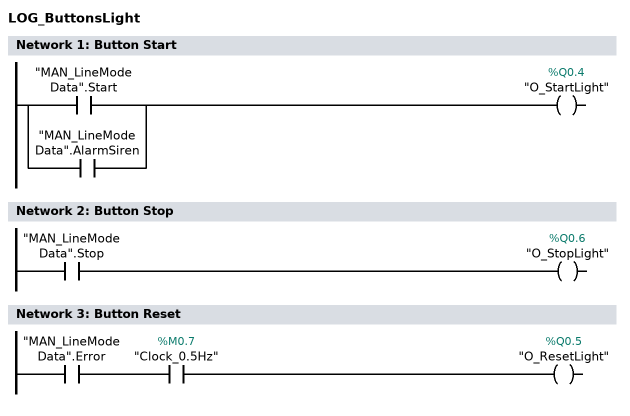
   RUNG wire#powerrail
      Contact( "MAN_LineModeData".Start )
      wire#w1
      Coil( "O_StartLight" )
   END_RUNG
   RUNG wire#powerrail
      Contact( "MAN_LineModeData".AlarmSiren )
   END_RUNG wire#w1
   // the same network as SCL:
   "O_StartLight" := "MAN_LineModeData".Start OR "MAN_LineModeData".AlarmSiren;
END_REGION

REGION Network 2: Button Stop
   RUNG wire#powerrail
      Contact( "MAN_LineModeData".Stop )
      Coil( "O_StopLight" )
   END_RUNG
   // the same network as SCL:
   "O_StopLight" := "MAN_LineModeData".Stop;
END_REGION

REGION Network 3: Button Reset
   RUNG wire#powerrail
      Contact( "MAN_LineModeData".Error )
      Contact( "Clock_0.5Hz" )
      Coil( "O_ResetLight" )
   END_RUNG
   // the same network as SCL:
   "O_ResetLight" := "MAN_LineModeData".Error AND "Clock_0.5Hz";
END_REGION
END_FUNCTION

FUNCTION "LOG_ButtonsManualLight" : Void   // FC15, LAD
{ S7_Optimized_Access := 'TRUE' }
VERSION : 0.1
// stored: AutoNumber true, IsIECCheckEnabled false, SetENOAutomatically false, UDAEnableTagReadback false
BEGIN

REGION Network 1: Button C1 light
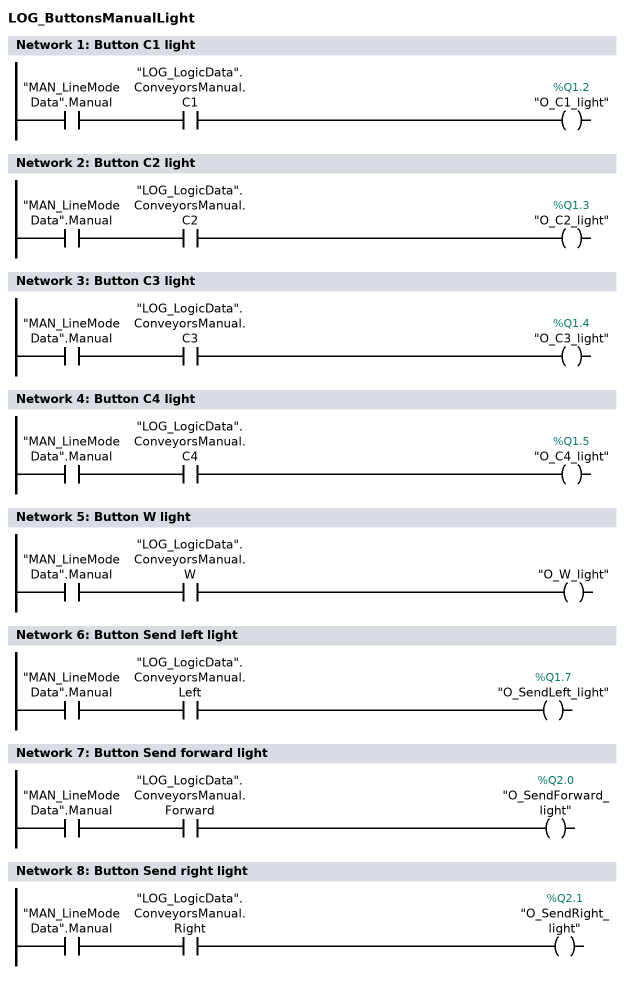
   RUNG wire#powerrail
      Contact( "MAN_LineModeData".Manual )
      Contact( "LOG_LogicData".ConveyorsManual.C1 )
      Coil( "O_C1_light" )
   END_RUNG
   // the same network as SCL:
   "O_C1_light" := "MAN_LineModeData".Manual AND "LOG_LogicData".ConveyorsManual.C1;
END_REGION

REGION Network 2: Button C2 light
   RUNG wire#powerrail
      Contact( "MAN_LineModeData".Manual )
      Contact( "LOG_LogicData".ConveyorsManual.C2 )
      Coil( "O_C2_light" )
   END_RUNG
   // the same network as SCL:
   "O_C2_light" := "MAN_LineModeData".Manual AND "LOG_LogicData".ConveyorsManual.C2;
END_REGION

REGION Network 3: Button C3 light
   RUNG wire#powerrail
      Contact( "MAN_LineModeData".Manual )
      Contact( "LOG_LogicData".ConveyorsManual.C3 )
      Coil( "O_C3_light" )
   END_RUNG
   // the same network as SCL:
   "O_C3_light" := "MAN_LineModeData".Manual AND "LOG_LogicData".ConveyorsManual.C3;
END_REGION

REGION Network 4: Button C4 light
   RUNG wire#powerrail
      Contact( "MAN_LineModeData".Manual )
      Contact( "LOG_LogicData".ConveyorsManual.C4 )
      Coil( "O_C4_light" )
   END_RUNG
   // the same network as SCL:
   "O_C4_light" := "MAN_LineModeData".Manual AND "LOG_LogicData".ConveyorsManual.C4;
END_REGION

REGION Network 5: Button W light
   RUNG wire#powerrail
      Contact( "MAN_LineModeData".Manual )
      Contact( "LOG_LogicData".ConveyorsManual.W )
      Coil( "O_W_light" )
   END_RUNG
   // the same network as SCL:
   "O_W_light" := "MAN_LineModeData".Manual AND "LOG_LogicData".ConveyorsManual.W;
END_REGION

REGION Network 6: Button Send left light
   RUNG wire#powerrail
      Contact( "MAN_LineModeData".Manual )
      Contact( "LOG_LogicData".ConveyorsManual.Left )
      Coil( "O_SendLeft_light" )
   END_RUNG
   // the same network as SCL:
   "O_SendLeft_light" := "MAN_LineModeData".Manual AND "LOG_LogicData".ConveyorsManual.Left;
END_REGION

REGION Network 7: Button Send forward light
   RUNG wire#powerrail
      Contact( "MAN_LineModeData".Manual )
      Contact( "LOG_LogicData".ConveyorsManual.Forward )
      Coil( "O_SendForward_light" )
   END_RUNG
   // the same network as SCL:
   "O_SendForward_light" := "MAN_LineModeData".Manual AND "LOG_LogicData".ConveyorsManual.Forward;
END_REGION

REGION Network 8: Button Send right light
   RUNG wire#powerrail
      Contact( "MAN_LineModeData".Manual )
      Contact( "LOG_LogicData".ConveyorsManual.Right )
      Coil( "O_SendRight_light" )
   END_RUNG
   // the same network as SCL:
   "O_SendRight_light" := "MAN_LineModeData".Manual AND "LOG_LogicData".ConveyorsManual.Right;
END_REGION
END_FUNCTION

FUNCTION "LOG_ColumnLight" : Void   // FC16, LAD
{ S7_Optimized_Access := 'TRUE' }
VERSION : 0.1
// stored: AutoNumber true, IsIECCheckEnabled false, SetENOAutomatically false, UDAEnableTagReadback false
   VAR_TEMP
      Green_1 : Bool;
      Green_2 : Bool;
      Yellow_1 : Bool;
      Yellow_2 : Bool;
   END_VAR
BEGIN

REGION Network 1: Start line manual mode signaling
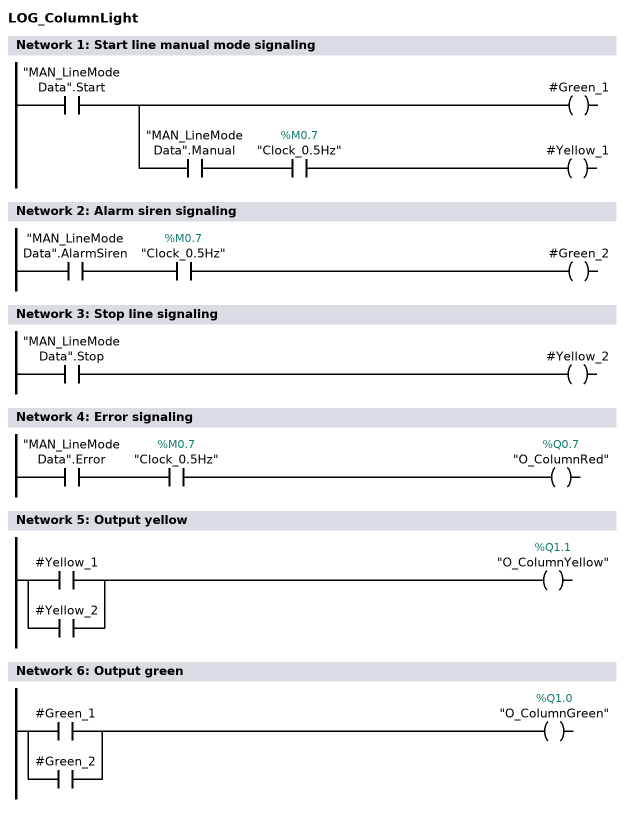
   RUNG wire#powerrail
      Contact( "MAN_LineModeData".Start )
      wire#w1
      Coil( #Green_1 )
   END_RUNG
   RUNG wire#w1
      Contact( "MAN_LineModeData".Manual )
      Contact( "Clock_0.5Hz" )
      Coil( #Yellow_1 )
   END_RUNG
   // the same network as SCL:
   #Green_1 := "MAN_LineModeData".Start;
   #Yellow_1 := "MAN_LineModeData".Start AND "MAN_LineModeData".Manual AND "Clock_0.5Hz";
END_REGION

REGION Network 2: Alarm siren signaling
   RUNG wire#powerrail
      Contact( "MAN_LineModeData".AlarmSiren )
      Contact( "Clock_0.5Hz" )
      Coil( #Green_2 )
   END_RUNG
   // the same network as SCL:
   #Green_2 := "MAN_LineModeData".AlarmSiren AND "Clock_0.5Hz";
END_REGION

REGION Network 3: Stop line signaling
   RUNG wire#powerrail
      Contact( "MAN_LineModeData".Stop )
      Coil( #Yellow_2 )
   END_RUNG
   // the same network as SCL:
   #Yellow_2 := "MAN_LineModeData".Stop;
END_REGION

REGION Network 4: Error signaling
   RUNG wire#powerrail
      Contact( "MAN_LineModeData".Error )
      Contact( "Clock_0.5Hz" )
      Coil( "O_ColumnRed" )
   END_RUNG
   // the same network as SCL:
   "O_ColumnRed" := "MAN_LineModeData".Error AND "Clock_0.5Hz";
END_REGION

REGION Network 5: Output yellow
   RUNG wire#powerrail
      Contact( #Yellow_1 )
      wire#w1
      Coil( "O_ColumnYellow" )
   END_RUNG
   RUNG wire#powerrail
      Contact( #Yellow_2 )
   END_RUNG wire#w1
   // the same network as SCL:
   "O_ColumnYellow" := #Yellow_1 OR #Yellow_2;
END_REGION

REGION Network 6: Output green
   RUNG wire#powerrail
      Contact( #Green_1 )
      wire#w1
      Coil( "O_ColumnGreen" )
   END_RUNG
   RUNG wire#powerrail
      Contact( #Green_2 )
   END_RUNG wire#w1
   // the same network as SCL:
   "O_ColumnGreen" := #Green_1 OR #Green_2;
END_REGION
END_FUNCTION

FUNCTION "LOG_Light" : Void   // FC11, LAD
{ S7_Optimized_Access := 'TRUE' }
VERSION : 0.1
// stored: AutoNumber true, IsIECCheckEnabled false, SetENOAutomatically false, UDAEnableTagReadback false
BEGIN

REGION Network 1: Call: ButtonsLight
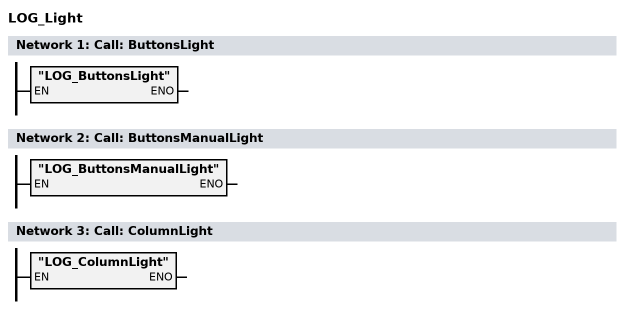
   RUNG wire#powerrail
      "LOG_ButtonsLight"()
   END_RUNG
   // the same network as SCL:
   "LOG_ButtonsLight"();
END_REGION

REGION Network 2: Call: ButtonsManualLight
   RUNG wire#powerrail
      "LOG_ButtonsManualLight"()
   END_RUNG
   // the same network as SCL:
   "LOG_ButtonsManualLight"();
END_REGION

REGION Network 3: Call: ColumnLight
   RUNG wire#powerrail
      "LOG_ColumnLight"()
   END_RUNG
   // the same network as SCL:
   "LOG_ColumnLight"();
END_REGION
END_FUNCTION

FUNCTION "LOG_Statistic" : Void   // FC8, LAD
{ S7_Optimized_Access := 'TRUE' }
VERSION : 0.1
// stored: AutoNumber false, IsIECCheckEnabled false, SetENOAutomatically false, UDAEnableTagReadback false
   VAR_TEMP
      t_RisingEdge : Bool;
   END_VAR
BEGIN

REGION Network 1: Call: CountPackages
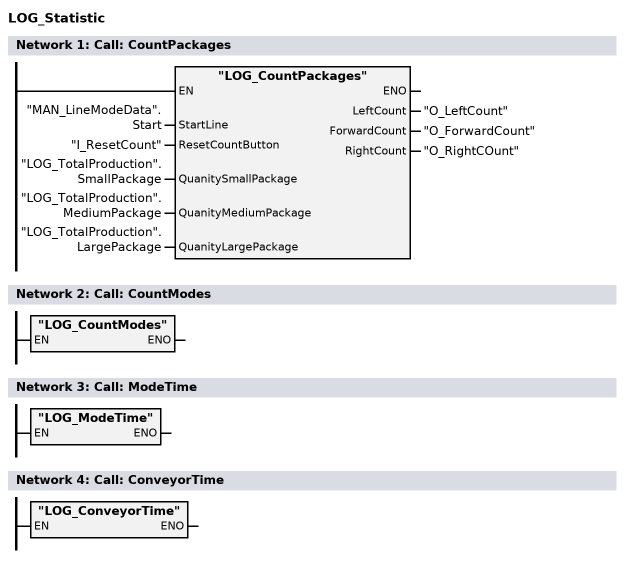
   RUNG wire#powerrail
      "LOG_CountPackages"(StartLine := "MAN_LineModeData".Start, ResetCountButton := "I_ResetCount", QuanitySmallPackage := "LOG_TotalProduction".SmallPackage, QuanityMediumPackage := "LOG_TotalProduction".MediumPackage, QuanityLargePackage := "LOG_TotalProduction".LargePackage, LeftCount => "O_LeftCount", ForwardCount => "O_ForwardCount", RightCount => "O_RightCOunt")
   END_RUNG
   // the same network as SCL:
   "LOG_CountPackages"(StartLine := "MAN_LineModeData".Start,
                       ResetCountButton := "I_ResetCount",
                       QuanitySmallPackage := "LOG_TotalProduction".SmallPackage,
                       QuanityMediumPackage := "LOG_TotalProduction".MediumPackage,
                       QuanityLargePackage := "LOG_TotalProduction".LargePackage,
                       LeftCount => "O_LeftCount",
                       ForwardCount => "O_ForwardCount",
                       RightCount => "O_RightCOunt");
END_REGION

REGION Network 2: Call: CountModes
   RUNG wire#powerrail
      "LOG_CountModes"()
   END_RUNG
   // the same network as SCL:
   "LOG_CountModes"();
END_REGION

REGION Network 3: Call: ModeTime
   RUNG wire#powerrail
      "LOG_ModeTime"()
   END_RUNG
   // the same network as SCL:
   "LOG_ModeTime"();
END_REGION

REGION Network 4: Call: ConveyorTime
   RUNG wire#powerrail
      "LOG_ConveyorTime"()
   END_RUNG
   // the same network as SCL:
   "LOG_ConveyorTime"();
END_REGION
END_FUNCTION

FUNCTION "LOG_CountPackages" : Void   // FC9, LAD
{ S7_Optimized_Access := 'TRUE' }
VERSION : 0.1
// stored: AutoNumber false, IsIECCheckEnabled false, SetENOAutomatically false, UDAEnableTagReadback false
   VAR_INPUT
      StartLine : Bool;
      ResetCountButton : Bool;
   END_VAR
   VAR_OUTPUT
      LeftCount : Int;
      ForwardCount : Int;
      RightCount : Int;
   END_VAR
   VAR_IN_OUT
      QuanitySmallPackage : Int;
      QuanityMediumPackage : Int;
      QuanityLargePackage : Int;
   END_VAR
BEGIN

REGION Network 1
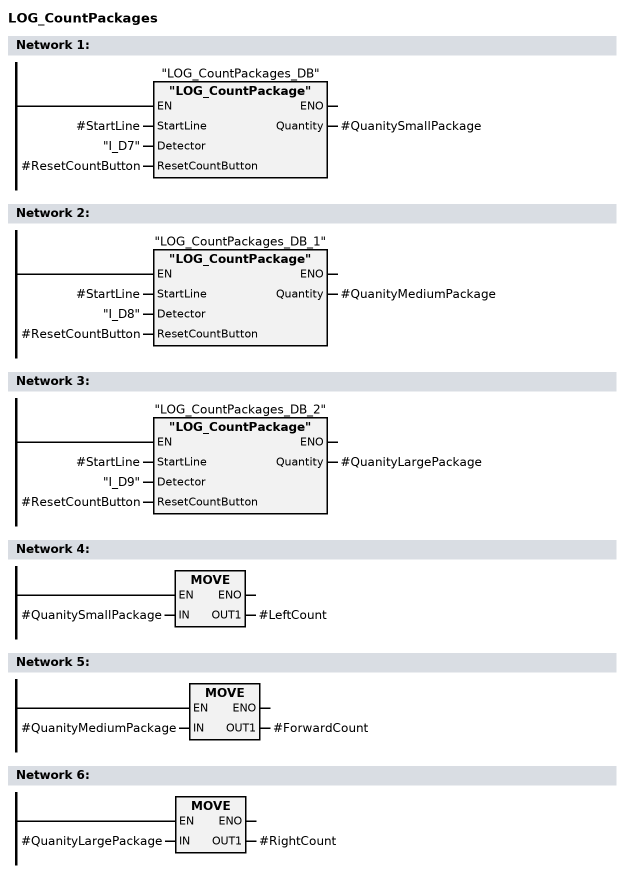
   RUNG wire#powerrail
      "LOG_CountPackages_DB"(StartLine := #StartLine, Detector := "I_D7", ResetCountButton := #ResetCountButton, Quantity => #QuanitySmallPackage)
   END_RUNG
   // the same network as SCL:
   "LOG_CountPackages_DB"(StartLine := #StartLine,   // "LOG_CountPackage"
                          Detector := "I_D7",
                          ResetCountButton := #ResetCountButton,
                          Quantity => #QuanitySmallPackage);
END_REGION

REGION Network 2
   RUNG wire#powerrail
      "LOG_CountPackages_DB_1"(StartLine := #StartLine, Detector := "I_D8", ResetCountButton := #ResetCountButton, Quantity => #QuanityMediumPackage)
   END_RUNG
   // the same network as SCL:
   "LOG_CountPackages_DB_1"(StartLine := #StartLine,   // "LOG_CountPackage"
                           Detector := "I_D8",
                           ResetCountButton := #ResetCountButton,
                           Quantity => #QuanityMediumPackage);
END_REGION

REGION Network 3
   RUNG wire#powerrail
      "LOG_CountPackages_DB_2"(StartLine := #StartLine, Detector := "I_D9", ResetCountButton := #ResetCountButton, Quantity => #QuanityLargePackage)
   END_RUNG
   // the same network as SCL:
   "LOG_CountPackages_DB_2"(StartLine := #StartLine,   // "LOG_CountPackage"
                           Detector := "I_D9",
                           ResetCountButton := #ResetCountButton,
                           Quantity => #QuanityLargePackage);
END_REGION

REGION Network 4
   RUNG wire#powerrail
      Move(in := #QuanitySmallPackage, out1 => #LeftCount)
   END_RUNG
   // the same network as SCL:
   #LeftCount := #QuanitySmallPackage;
END_REGION

REGION Network 5
   RUNG wire#powerrail
      Move(in := #QuanityMediumPackage, out1 => #ForwardCount)
   END_RUNG
   // the same network as SCL:
   #ForwardCount := #QuanityMediumPackage;
END_REGION

REGION Network 6
   RUNG wire#powerrail
      Move(in := #QuanityLargePackage, out1 => #RightCount)
   END_RUNG
   // the same network as SCL:
   #RightCount := #QuanityLargePackage;
END_REGION
END_FUNCTION

FUNCTION_BLOCK "LOG_CountPackage"   // FB4, LAD
{ S7_Optimized_Access := 'TRUE' }
VERSION : 0.1
// stored: AutoNumber true, IsIECCheckEnabled false, IsRetainMemResEnabled false, MemoryReserve 100, SetENOAutomatically false, UDAEnableTagReadback false
   VAR_INPUT
      StartLine : Bool;
      Detector : Bool;
      ResetCountButton : Bool;
   END_VAR
   VAR_OUTPUT
      Quantity : Int;
   END_VAR
   VAR RETAIN
      IEC_Counter_0_Instance { ExternalAccessible := 'False'; ExternalVisible := 'False'; ExternalWritable := 'False'} : CTU_INT;
      N_Detector { S7_SetPoint := 'True'} : Bool;
   END_VAR
   VAR_TEMP   // added for the SCL form of the ladder/FBD networks
      _w1 : Bool;
   END_VAR
BEGIN

REGION Network 1
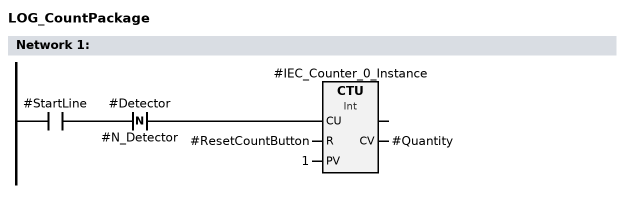
   RUNG wire#powerrail
      Contact( #StartLine )
      N_Contact(operand := #Detector, bit := #N_Detector)
      { S7_Templates := "value_type := Int" } #IEC_Counter_0_Instance.CTU(r := #ResetCountButton, pv := 1, cv => #Quantity)
   END_RUNG
   // the same network as SCL:
   #_w1 := #StartLine AND NOT #Detector AND #N_Detector;   // falling edge of #Detector
   #N_Detector := #Detector;
   #IEC_Counter_0_Instance(CU := #_w1, R := #ResetCountButton, PV := 1, CV => #Quantity);   // CTU
END_REGION
END_FUNCTION_BLOCK

FUNCTION "LOG_CountModes" : Void   // FC19, LAD
{ S7_Optimized_Access := 'TRUE' }
VERSION : 0.1
// stored: AutoNumber true, IsIECCheckEnabled false, SetENOAutomatically false, UDAEnableTagReadback false
BEGIN

REGION Network 1: Call: CountMode - Auto
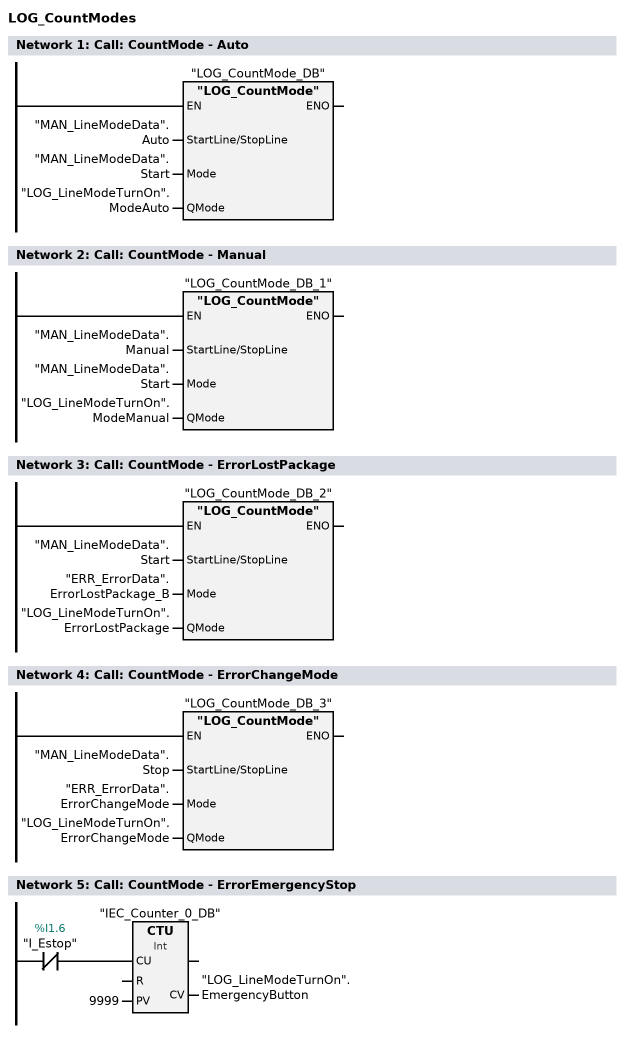
   RUNG wire#powerrail
      "LOG_CountMode_DB"("StartLine/StopLine" := "MAN_LineModeData".Auto, Mode := "MAN_LineModeData".Start, QMode := "LOG_LineModeTurnOn".ModeAuto)
   END_RUNG
   // the same network as SCL:
   "LOG_CountMode_DB"("StartLine/StopLine" := "MAN_LineModeData".Auto,   // "LOG_CountMode"
                      Mode := "MAN_LineModeData".Start,
                      QMode := "LOG_LineModeTurnOn".ModeAuto);
END_REGION

REGION Network 2: Call: CountMode - Manual
   RUNG wire#powerrail
      "LOG_CountMode_DB_1"("StartLine/StopLine" := "MAN_LineModeData".Manual, Mode := "MAN_LineModeData".Start, QMode := "LOG_LineModeTurnOn".ModeManual)
   END_RUNG
   // the same network as SCL:
   "LOG_CountMode_DB_1"("StartLine/StopLine" := "MAN_LineModeData".Manual,   // "LOG_CountMode"
                        Mode := "MAN_LineModeData".Start,
                        QMode := "LOG_LineModeTurnOn".ModeManual);
END_REGION

REGION Network 3: Call: CountMode - ErrorLostPackage
   RUNG wire#powerrail
      "LOG_CountMode_DB_2"("StartLine/StopLine" := "MAN_LineModeData".Start, Mode := "ERR_ErrorData".ErrorLostPackage_B, QMode := "LOG_LineModeTurnOn".ErrorLostPackage)
   END_RUNG
   // the same network as SCL:
   "LOG_CountMode_DB_2"("StartLine/StopLine" := "MAN_LineModeData".Start,   // "LOG_CountMode"
                        Mode := "ERR_ErrorData".ErrorLostPackage_B,
                        QMode := "LOG_LineModeTurnOn".ErrorLostPackage);
END_REGION

REGION Network 4: Call: CountMode - ErrorChangeMode
   RUNG wire#powerrail
      "LOG_CountMode_DB_3"("StartLine/StopLine" := "MAN_LineModeData".Stop, Mode := "ERR_ErrorData".ErrorChangeMode, QMode := "LOG_LineModeTurnOn".ErrorChangeMode)
   END_RUNG
   // the same network as SCL:
   "LOG_CountMode_DB_3"("StartLine/StopLine" := "MAN_LineModeData".Stop,   // "LOG_CountMode"
                        Mode := "ERR_ErrorData".ErrorChangeMode,
                        QMode := "LOG_LineModeTurnOn".ErrorChangeMode);
END_REGION

REGION Network 5: Call: CountMode - ErrorEmergencyStop
   RUNG wire#powerrail
      I_Contact( "I_Estop" )
      { S7_Templates := "value_type := Int" } "IEC_Counter_0_DB".CTU(r :=, pv := 9999, cv => "LOG_LineModeTurnOn".EmergencyButton)
   END_RUNG
   // the same network as SCL:
   "IEC_Counter_0_DB".CTU(CU := NOT "I_Estop", PV := 9999, CV => "LOG_LineModeTurnOn".EmergencyButton);
END_REGION
END_FUNCTION

FUNCTION_BLOCK "LOG_CountMode"   // FB3, LAD
{ S7_Optimized_Access := 'TRUE' }
VERSION : 0.1
// stored: AutoNumber true, IsIECCheckEnabled false, IsRetainMemResEnabled false, MemoryReserve 100, SetENOAutomatically false, UDAEnableTagReadback false
   VAR_INPUT
      "StartLine/StopLine" : Bool;
      Mode : Bool;
   END_VAR
   VAR_IN_OUT
      QMode : UDInt;
   END_VAR
   VAR
      P_Mode : Bool;
   END_VAR
   VAR_TEMP   // added for the SCL form of the ladder/FBD networks
      _w1 : Bool;
   END_VAR
BEGIN

REGION Network 1
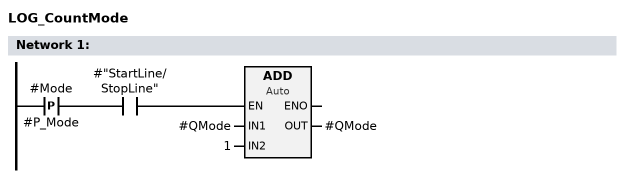
   RUNG wire#powerrail
      P_Contact(operand := #Mode, bit := #P_Mode)
      Contact( #"StartLine/StopLine" )
      { S7_GenerateENO := "TRUE" } Add(in1 := #QMode, in2 := 1, out => #QMode)
   END_RUNG
   // the same network as SCL:
   #_w1 := #Mode AND NOT #P_Mode;   // rising edge of #Mode
   #P_Mode := #Mode;
   IF #_w1 AND #"StartLine/StopLine" THEN #QMode := #QMode + 1; END_IF;
END_REGION
END_FUNCTION_BLOCK

FUNCTION "LOG_ModeTime" : Void   // FC18, LAD
{ S7_Optimized_Access := 'TRUE' }
VERSION : 0.1
// stored: AutoNumber true, IsIECCheckEnabled false, SetENOAutomatically false, UDAEnableTagReadback false
   VAR_TEMP
      t_RisingEdge : Bool;
   END_VAR
BEGIN

REGION Network 1: Trigger
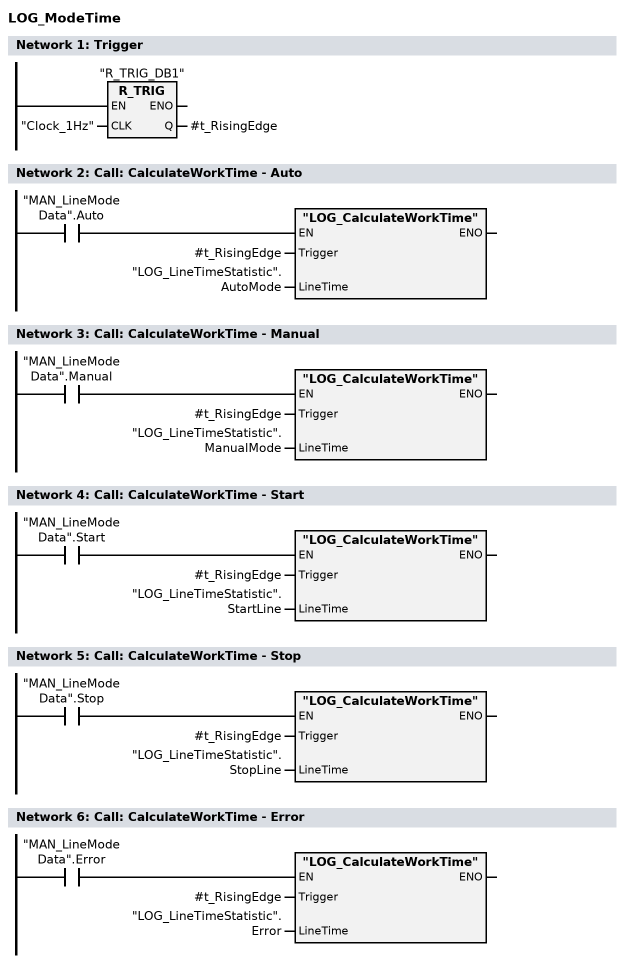
   RUNG wire#powerrail
      "R_TRIG_DB1".R_TRIG(CLK := "Clock_1Hz", Q => #t_RisingEdge)
   END_RUNG
   // the same network as SCL:
   "R_TRIG_DB1"(CLK := "Clock_1Hz", Q => #t_RisingEdge);   // R_TRIG
END_REGION

REGION Network 2: Call: CalculateWorkTime - Auto
   RUNG wire#powerrail
      Contact( "MAN_LineModeData".Auto )
      "LOG_CalculateWorkTime"(Trigger := #t_RisingEdge, LineTime := "LOG_LineTimeStatistic".AutoMode)
   END_RUNG
   // the same network as SCL:
   IF "MAN_LineModeData".Auto THEN
       "LOG_CalculateWorkTime"(Trigger := #t_RisingEdge, LineTime := "LOG_LineTimeStatistic".AutoMode);
   END_IF;
END_REGION

REGION Network 3: Call: CalculateWorkTime - Manual
   RUNG wire#powerrail
      Contact( "MAN_LineModeData".Manual )
      "LOG_CalculateWorkTime"(Trigger := #t_RisingEdge, LineTime := "LOG_LineTimeStatistic".ManualMode)
   END_RUNG
   // the same network as SCL:
   IF "MAN_LineModeData".Manual THEN
       "LOG_CalculateWorkTime"(Trigger := #t_RisingEdge, LineTime := "LOG_LineTimeStatistic".ManualMode);
   END_IF;
END_REGION

REGION Network 4: Call: CalculateWorkTime - Start
   RUNG wire#powerrail
      Contact( "MAN_LineModeData".Start )
      "LOG_CalculateWorkTime"(Trigger := #t_RisingEdge, LineTime := "LOG_LineTimeStatistic".StartLine)
   END_RUNG
   // the same network as SCL:
   IF "MAN_LineModeData".Start THEN
       "LOG_CalculateWorkTime"(Trigger := #t_RisingEdge, LineTime := "LOG_LineTimeStatistic".StartLine);
   END_IF;
END_REGION

REGION Network 5: Call: CalculateWorkTime - Stop
   RUNG wire#powerrail
      Contact( "MAN_LineModeData".Stop )
      "LOG_CalculateWorkTime"(Trigger := #t_RisingEdge, LineTime := "LOG_LineTimeStatistic".StopLine)
   END_RUNG
   // the same network as SCL:
   IF "MAN_LineModeData".Stop THEN
       "LOG_CalculateWorkTime"(Trigger := #t_RisingEdge, LineTime := "LOG_LineTimeStatistic".StopLine);
   END_IF;
END_REGION

REGION Network 6: Call: CalculateWorkTime - Error
   RUNG wire#powerrail
      Contact( "MAN_LineModeData".Error )
      "LOG_CalculateWorkTime"(Trigger := #t_RisingEdge, LineTime := "LOG_LineTimeStatistic".Error)
   END_RUNG
   // the same network as SCL:
   IF "MAN_LineModeData".Error THEN
       "LOG_CalculateWorkTime"(Trigger := #t_RisingEdge, LineTime := "LOG_LineTimeStatistic".Error);
   END_IF;
END_REGION
END_FUNCTION

FUNCTION "LOG_CalculateWorkTime" : Void   // FC1300, LAD
{ S7_Optimized_Access := 'TRUE' }
VERSION : 0.1
// stored: AutoNumber false, IsIECCheckEnabled false, SetENOAutomatically false, UDAEnableTagReadback false
   VAR_INPUT
      Trigger : Bool;
   END_VAR
   VAR_IN_OUT
      LineTime : "stt_TimeWork";
   END_VAR
   VAR_TEMP   // added for the SCL form of the ladder/FBD networks
      _w1 : Bool;
   END_VAR
BEGIN

REGION Network 1: Seconds
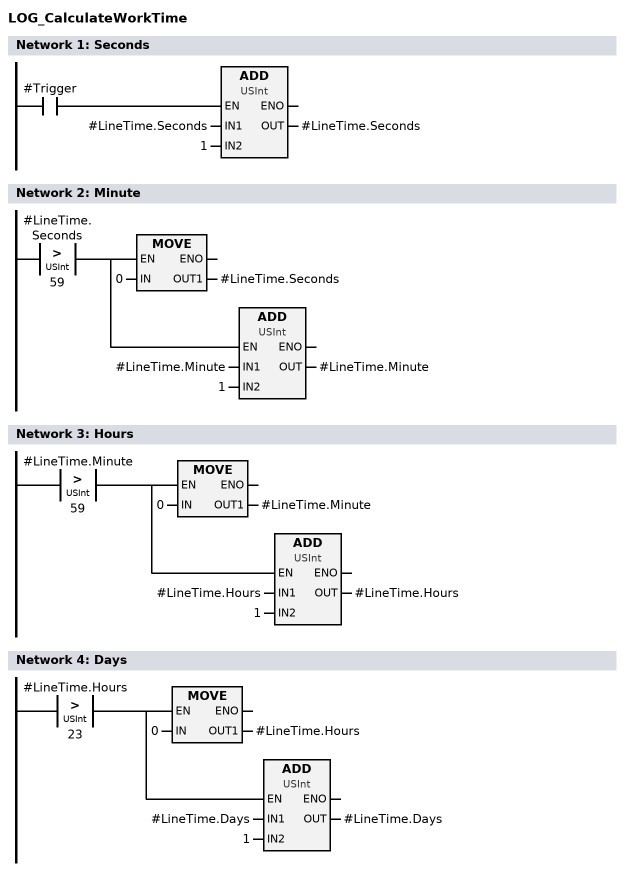
   RUNG wire#powerrail
      Contact( #Trigger )
      { S7_Templates := "SrcType := USInt"; S7_GenerateENO := "TRUE" } Add(in1 := #LineTime.Seconds, in2 := 1, out => #LineTime.Seconds)
   END_RUNG
   // the same network as SCL:
   IF #Trigger THEN #LineTime.Seconds := #LineTime.Seconds + 1; END_IF;
END_REGION

REGION Network 2: Minute
   RUNG wire#powerrail
      { S7_Templates := "SrcType := USInt" } GT_Contact(in1 := #LineTime.Seconds, in2 := 59)
      wire#w1
      { S7_GenerateENO := "TRUE" } Move(in := 0, out1 => #LineTime.Seconds)
   END_RUNG
   RUNG wire#w1
      { S7_Templates := "SrcType := USInt"; S7_GenerateENO := "TRUE" } Add(in1 := #LineTime.Minute, in2 := 1, out => #LineTime.Minute)
   END_RUNG
   // the same network as SCL:
   #_w1 := #LineTime.Seconds > 59;
   IF #_w1 THEN
       #LineTime.Seconds := 0;
       #LineTime.Minute := #LineTime.Minute + 1;
   END_IF;
END_REGION

REGION Network 3: Hours
   RUNG wire#powerrail
      { S7_Templates := "SrcType := USInt" } GT_Contact(in1 := #LineTime.Minute, in2 := 59)
      wire#w1
      { S7_GenerateENO := "TRUE" } Move(in := 0, out1 => #LineTime.Minute)
   END_RUNG
   RUNG wire#w1
      { S7_Templates := "SrcType := USInt"; S7_GenerateENO := "TRUE" } Add(in1 := #LineTime.Hours, in2 := 1, out => #LineTime.Hours)
   END_RUNG
   // the same network as SCL:
   #_w1 := #LineTime.Minute > 59;
   IF #_w1 THEN
       #LineTime.Minute := 0;
       #LineTime.Hours := #LineTime.Hours + 1;
   END_IF;
END_REGION

REGION Network 4: Days
   RUNG wire#powerrail
      { S7_Templates := "SrcType := USInt" } GT_Contact(in1 := #LineTime.Hours, in2 := 23)
      wire#w1
      { S7_GenerateENO := "TRUE" } Move(in := 0, out1 => #LineTime.Hours)
   END_RUNG
   RUNG wire#w1
      { S7_Templates := "SrcType := USInt"; S7_GenerateENO := "TRUE" } Add(in1 := #LineTime.Days, in2 := 1, out => #LineTime.Days)
   END_RUNG
   // the same network as SCL:
   #_w1 := #LineTime.Hours > 23;
   IF #_w1 THEN
       #LineTime.Hours := 0;
       #LineTime.Days := #LineTime.Days + 1;
   END_IF;
END_REGION
END_FUNCTION

FUNCTION "LOG_ConveyorTime" : Void   // FC20, LAD
{ S7_Optimized_Access := 'TRUE' }
VERSION : 0.1
// stored: AutoNumber true, IsIECCheckEnabled false, SetENOAutomatically false, UDAEnableTagReadback false
   VAR_TEMP
      t_RisingTime : Bool;
   END_VAR
BEGIN

REGION Network 1: Trigger
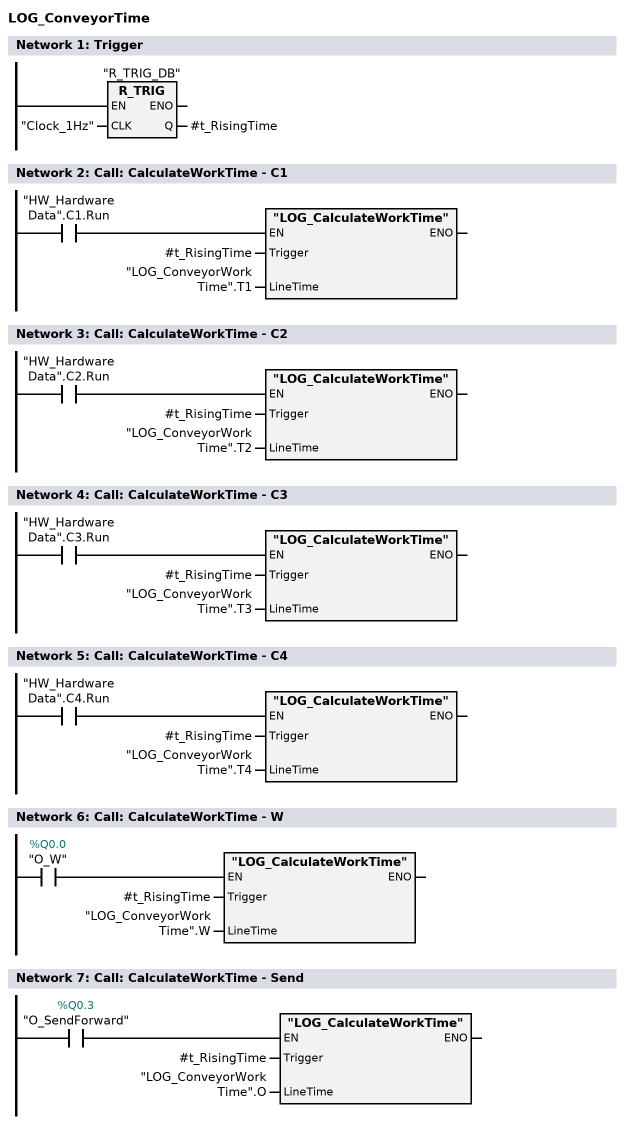
   RUNG wire#powerrail
      "R_TRIG_DB".R_TRIG(CLK := "Clock_1Hz", Q => #t_RisingTime)
   END_RUNG
   // the same network as SCL:
   "R_TRIG_DB"(CLK := "Clock_1Hz", Q => #t_RisingTime);   // R_TRIG
END_REGION

REGION Network 2: Call: CalculateWorkTime - C1
   RUNG wire#powerrail
      Contact( "HW_HardwareData".C1.Run )
      "LOG_CalculateWorkTime"(Trigger := #t_RisingTime, LineTime := "LOG_ConveyorWorkTime".T1)
   END_RUNG
   // the same network as SCL:
   IF "HW_HardwareData".C1.Run THEN
       "LOG_CalculateWorkTime"(Trigger := #t_RisingTime, LineTime := "LOG_ConveyorWorkTime".T1);
   END_IF;
END_REGION

REGION Network 3: Call: CalculateWorkTime - C2
   RUNG wire#powerrail
      Contact( "HW_HardwareData".C2.Run )
      "LOG_CalculateWorkTime"(Trigger := #t_RisingTime, LineTime := "LOG_ConveyorWorkTime".T2)
   END_RUNG
   // the same network as SCL:
   IF "HW_HardwareData".C2.Run THEN
       "LOG_CalculateWorkTime"(Trigger := #t_RisingTime, LineTime := "LOG_ConveyorWorkTime".T2);
   END_IF;
END_REGION

REGION Network 4: Call: CalculateWorkTime - C3
   RUNG wire#powerrail
      Contact( "HW_HardwareData".C3.Run )
      "LOG_CalculateWorkTime"(Trigger := #t_RisingTime, LineTime := "LOG_ConveyorWorkTime".T3)
   END_RUNG
   // the same network as SCL:
   IF "HW_HardwareData".C3.Run THEN
       "LOG_CalculateWorkTime"(Trigger := #t_RisingTime, LineTime := "LOG_ConveyorWorkTime".T3);
   END_IF;
END_REGION

REGION Network 5: Call: CalculateWorkTime - C4
   RUNG wire#powerrail
      Contact( "HW_HardwareData".C4.Run )
      "LOG_CalculateWorkTime"(Trigger := #t_RisingTime, LineTime := "LOG_ConveyorWorkTime".T4)
   END_RUNG
   // the same network as SCL:
   IF "HW_HardwareData".C4.Run THEN
       "LOG_CalculateWorkTime"(Trigger := #t_RisingTime, LineTime := "LOG_ConveyorWorkTime".T4);
   END_IF;
END_REGION

REGION Network 6: Call: CalculateWorkTime - W
   RUNG wire#powerrail
      Contact( "O_W" )
      "LOG_CalculateWorkTime"(Trigger := #t_RisingTime, LineTime := "LOG_ConveyorWorkTime".W)
   END_RUNG
   // the same network as SCL:
   IF "O_W" THEN
       "LOG_CalculateWorkTime"(Trigger := #t_RisingTime, LineTime := "LOG_ConveyorWorkTime".W);
   END_IF;
END_REGION

REGION Network 7: Call: CalculateWorkTime - Send
   RUNG wire#powerrail
      Contact( "O_SendForward" )
      "LOG_CalculateWorkTime"(Trigger := #t_RisingTime, LineTime := "LOG_ConveyorWorkTime".O)
   END_RUNG
   // the same network as SCL:
   IF "O_SendForward" THEN
       "LOG_CalculateWorkTime"(Trigger := #t_RisingTime, LineTime := "LOG_ConveyorWorkTime".O);
   END_IF;
END_REGION
END_FUNCTION

DATA_BLOCK "ERR_ChangeMode_DB"   // DB23
VERSION : 0.1
// stored: AutoNumber true, InstanceOfName ERR_ChangeMode, InstanceOfType FB
"ERR_ChangeMode"
BEGIN
END_DATA_BLOCK

DATA_BLOCK "ERR_EStop_DB"   // DB21
VERSION : 0.1
// stored: AutoNumber true, InstanceOfName ERR_EStop, InstanceOfType FB
"ERR_EStop"
BEGIN
END_DATA_BLOCK

DATA_BLOCK "HW_MotorControle_DB"   // DB6
VERSION : 0.1
// stored: AutoNumber true, InstanceOfName HW_MotorControle, InstanceOfType FB
"HW_MotorControle"
BEGIN
END_DATA_BLOCK

DATA_BLOCK "HW_MotorControle_DB_1"   // DB8
VERSION : 0.1
// stored: AutoNumber true, InstanceOfName HW_MotorControle, InstanceOfType FB
"HW_MotorControle"
BEGIN
END_DATA_BLOCK

DATA_BLOCK "HW_MotorControle_DB_2"   // DB9
VERSION : 0.1
// stored: AutoNumber true, InstanceOfName HW_MotorControle, InstanceOfType FB
"HW_MotorControle"
BEGIN
END_DATA_BLOCK

DATA_BLOCK "HW_MotorControle_DB_3"   // DB10
VERSION : 0.1
// stored: AutoNumber true, InstanceOfName HW_MotorControle, InstanceOfType FB
"HW_MotorControle"
BEGIN
END_DATA_BLOCK

DATA_BLOCK "HW_MovingAverageFilter_DB"   // DB3
VERSION : 0.1
// stored: AutoNumber true, InstanceOfName HW_MovingAverageFilter, InstanceOfType FB
"HW_MovingAverageFilter"
BEGIN
END_DATA_BLOCK

DATA_BLOCK "IEC_Counter_0_DB"   // DB35
{ S7_Optimized_Access := 'TRUE' }
// stored: AutoNumber true, InstanceOfName IEC_COUNTER, OfSystemLibElement IEC_COUNTER, OfSystemLibVersion 1.0
"IEC_COUNTER"
   // VAR RETAIN
   //    CU : Bool;
   //    CD : Bool;
   //    R : Bool;
   //    LD : Bool;
   //    QU : Bool;
   //    QD : Bool;
   //    PV : Int;
   //    CV : Int;
   // END_VAR
BEGIN
END_DATA_BLOCK

DATA_BLOCK "LOG_AutoControle_DB"   // DB11
VERSION : 0.1
// stored: AutoNumber true, InstanceOfName LOG_AutoControle, InstanceOfType FB
"LOG_AutoControle"
BEGIN
END_DATA_BLOCK

DATA_BLOCK "LOG_CountMode_DB"   // DB31
VERSION : 0.1
// stored: AutoNumber true, InstanceOfName LOG_CountMode, InstanceOfType FB
"LOG_CountMode"
BEGIN
END_DATA_BLOCK

DATA_BLOCK "LOG_CountMode_DB_1"   // DB32
VERSION : 0.1
// stored: AutoNumber true, InstanceOfName LOG_CountMode, InstanceOfType FB
"LOG_CountMode"
BEGIN
END_DATA_BLOCK

DATA_BLOCK "LOG_CountMode_DB_2"   // DB33
VERSION : 0.1
// stored: AutoNumber true, InstanceOfName LOG_CountMode, InstanceOfType FB
"LOG_CountMode"
BEGIN
END_DATA_BLOCK

DATA_BLOCK "LOG_CountMode_DB_3"   // DB34
VERSION : 0.1
// stored: AutoNumber true, InstanceOfName LOG_CountMode, InstanceOfType FB
"LOG_CountMode"
BEGIN
END_DATA_BLOCK

DATA_BLOCK "LOG_CountPackages_DB"   // DB36
VERSION : 0.1
// stored: AutoNumber true, InstanceOfName LOG_CountPackage, InstanceOfType FB
"LOG_CountPackage"
BEGIN
END_DATA_BLOCK

DATA_BLOCK "LOG_CountPackages_DB_1"   // DB37
VERSION : 0.1
// stored: AutoNumber true, InstanceOfName LOG_CountPackage, InstanceOfType FB
"LOG_CountPackage"
BEGIN
END_DATA_BLOCK

DATA_BLOCK "LOG_CountPackages_DB_2"   // DB38
VERSION : 0.1
// stored: AutoNumber true, InstanceOfName LOG_CountPackage, InstanceOfType FB
"LOG_CountPackage"
BEGIN
END_DATA_BLOCK

DATA_BLOCK "LOG_ManualModule_DB"   // DB12
VERSION : 0.1
// stored: AutoNumber true, InstanceOfName LOG_ManualModule, InstanceOfType FB
"LOG_ManualModule"
BEGIN
END_DATA_BLOCK

DATA_BLOCK "LOG_ManualModule_DB_1"   // DB13
VERSION : 0.1
// stored: AutoNumber true, InstanceOfName LOG_ManualModule, InstanceOfType FB
"LOG_ManualModule"
BEGIN
END_DATA_BLOCK

DATA_BLOCK "LOG_ManualModule_DB_2"   // DB14
VERSION : 0.1
// stored: AutoNumber true, InstanceOfName LOG_ManualModule, InstanceOfType FB
"LOG_ManualModule"
BEGIN
END_DATA_BLOCK

DATA_BLOCK "LOG_ManualModule_DB_3"   // DB15
VERSION : 0.1
// stored: AutoNumber true, InstanceOfName LOG_ManualModule, InstanceOfType FB
"LOG_ManualModule"
BEGIN
END_DATA_BLOCK

DATA_BLOCK "LOG_ManualModule_DB_4"   // DB17
VERSION : 0.1
// stored: AutoNumber true, InstanceOfName LOG_ManualModule, InstanceOfType FB
"LOG_ManualModule"
BEGIN
END_DATA_BLOCK

DATA_BLOCK "LOG_ManualModule_DB_5"   // DB18
VERSION : 0.1
// stored: AutoNumber true, InstanceOfName LOG_ManualModule, InstanceOfType FB
"LOG_ManualModule"
BEGIN
END_DATA_BLOCK

DATA_BLOCK "LOG_ManualModule_DB_6"   // DB19
VERSION : 0.1
// stored: AutoNumber true, InstanceOfName LOG_ManualModule, InstanceOfType FB
"LOG_ManualModule"
BEGIN
END_DATA_BLOCK

DATA_BLOCK "LOG_ManualModule_DB_7"   // DB20
VERSION : 0.1
// stored: AutoNumber true, InstanceOfName LOG_ManualModule, InstanceOfType FB
"LOG_ManualModule"
BEGIN
END_DATA_BLOCK

DATA_BLOCK "MAN_ControlLine_DB"   // DB2
VERSION : 0.1
// stored: AutoNumber true, InstanceOfName MAN_ControlLine, InstanceOfType FB
"MAN_ControlLine"
BEGIN
END_DATA_BLOCK

DATA_BLOCK "MAN_ControlLine_DB_1"   // DB5
VERSION : 0.1
// stored: AutoNumber true, InstanceOfName MAN_ControlLine, InstanceOfType FB
"MAN_ControlLine"
BEGIN
END_DATA_BLOCK

DATA_BLOCK "R_TRIG_DB"   // DB42
// stored: AutoNumber true, InstanceOfName R_TRIG, OfSystemLibElement R_TRIG, OfSystemLibVersion 1.0
"R_TRIG"
   // VAR_INPUT
   //    CLK : Bool;
   // END_VAR
   // VAR_OUTPUT
   //    Q : Bool;
   // END_VAR
   // VAR
   //    Stat_Bit : Bool;
   // END_VAR
BEGIN
END_DATA_BLOCK

DATA_BLOCK "R_TRIG_DB1"   // DB45
// stored: AutoNumber true, InstanceOfName R_TRIG, OfSystemLibElement R_TRIG, OfSystemLibVersion 1.0
"R_TRIG"
   // VAR_INPUT
   //    CLK : Bool;
   // END_VAR
   // VAR_OUTPUT
   //    Q : Bool;
   // END_VAR
   // VAR
   //    Stat_Bit : Bool;
   // END_VAR
BEGIN
END_DATA_BLOCK

DATA_BLOCK "ERR_LostPackage_DB"   // DB24
VERSION : 0.1
// stored: AutoNumber true, InstanceOfName ERR_LostPackage, InstanceOfType FB
"ERR_LostPackage"
BEGIN
END_DATA_BLOCK

DATA_BLOCK "ERR_LostPackage_DB_1"   // DB25
VERSION : 0.1
// stored: AutoNumber true, InstanceOfName ERR_LostPackage, InstanceOfType FB
"ERR_LostPackage"
BEGIN
END_DATA_BLOCK

DATA_BLOCK "ERR_LostPackage_DB_2"   // DB26
VERSION : 0.1
// stored: AutoNumber true, InstanceOfName ERR_LostPackage, InstanceOfType FB
"ERR_LostPackage"
BEGIN
END_DATA_BLOCK

DATA_BLOCK "ERR_LostPackage_DB_3"   // DB28
VERSION : 0.1
// stored: AutoNumber true, InstanceOfName ERR_LostPackage, InstanceOfType FB
"ERR_LostPackage"
BEGIN
END_DATA_BLOCK

DATA_BLOCK "ERR_LostPackage_DB_4"   // DB29
VERSION : 0.1
// stored: AutoNumber true, InstanceOfName ERR_LostPackage, InstanceOfType FB
"ERR_LostPackage"
BEGIN
END_DATA_BLOCK

DATA_BLOCK "ERR_LostPackage_DB_5"   // DB30
VERSION : 0.1
// stored: AutoNumber true, InstanceOfName ERR_LostPackage, InstanceOfType FB
"ERR_LostPackage"
BEGIN
END_DATA_BLOCK
